PROGRAM PRG_TEST
VAR
    _StringBuilder_Test : StringBuilder_Test;
END_VAR

TcUnit.RUN();

END_PROGRAM

(* stored: Version 1.1.0.1
   POU PRG_TEST: Id {89d6d83b-e661-4729-8376-220f86d31845}, SpecialFunc None *)
